// TIA Portal V20 export
// export: Created 2025-12-01T14:57:37.2453598Z, ExportSetting None, DisplayName Totally Integrated Automation Portal, DisplayVersion V20 Update 3, DisplayName TIA Portal Openness, DisplayVersion V20 Update 3, DisplayName TIA Portal Version Control Interface, DisplayVersion V20 Update 3, DisplayName STEP 7 Professional, DisplayVersion V20 Update 3, DisplayName STEP 7 Safety, DisplayVersion V20 Update 2, DisplayName WinCC Basic/Comfort/Advanced, DisplayVersion V20 Update 3, DisplayName WinCC Professional, DisplayVersion V20 Update 3, DisplayName WinCC Unified, DisplayVersion V20 Update 3
FUNCTION_BLOCK "FB74_Presion_DesPaletizadorCajasPlastico"   // FB74, LAD
TITLE = Calculo de la Presion del DesPaletizador de Cajas de Plastico
{ S7_Optimized_Access := 'FALSE' }
// stored: AutoNumber false, SetENOAutomatically false
   VAR_INPUT
      EstadoVI_Mesa : "EstadosMesa";
      EstadoVI_MesaSalida : "EstadosMesa";
      Mesa : UInt;
      MesaSalida : UInt;
      OrdenDesPaletizar : Bool;
      Abierta_PalaMovil : Bool;
      Abriendo_PalaMovil : Bool;
      Cerrando_PalaMovil : Bool;
   END_VAR
   VAR_OUTPUT
      PresionAnalogica : Word;
   END_VAR
   VAR
      TMPInicioPresion : UDInt;
      PresionCalculada : Word;
      MemoPresionSalida : Int;
      CalcularPresion : Bool;
      FinCalcularPresion : Bool;
      RecogerPresion : Bool;
   END_VAR
   VAR_TEMP
      PresionAConvertir : Int;
      PresionSalida : Word;
      PresionDef_Cerrar : Word;
      PresionDef_Abrir : Word;
      PresionInicialCerrar : Int;
      V_TMPInicioPresion : UDInt;
      OK_InicioPresion : Bool;
   END_VAR
   VAR_TEMP   // added for the SCL form of the ladder/FBD networks
      _w1 : Bool;
   END_VAR
BEGIN

REGION Network 1: Incializar
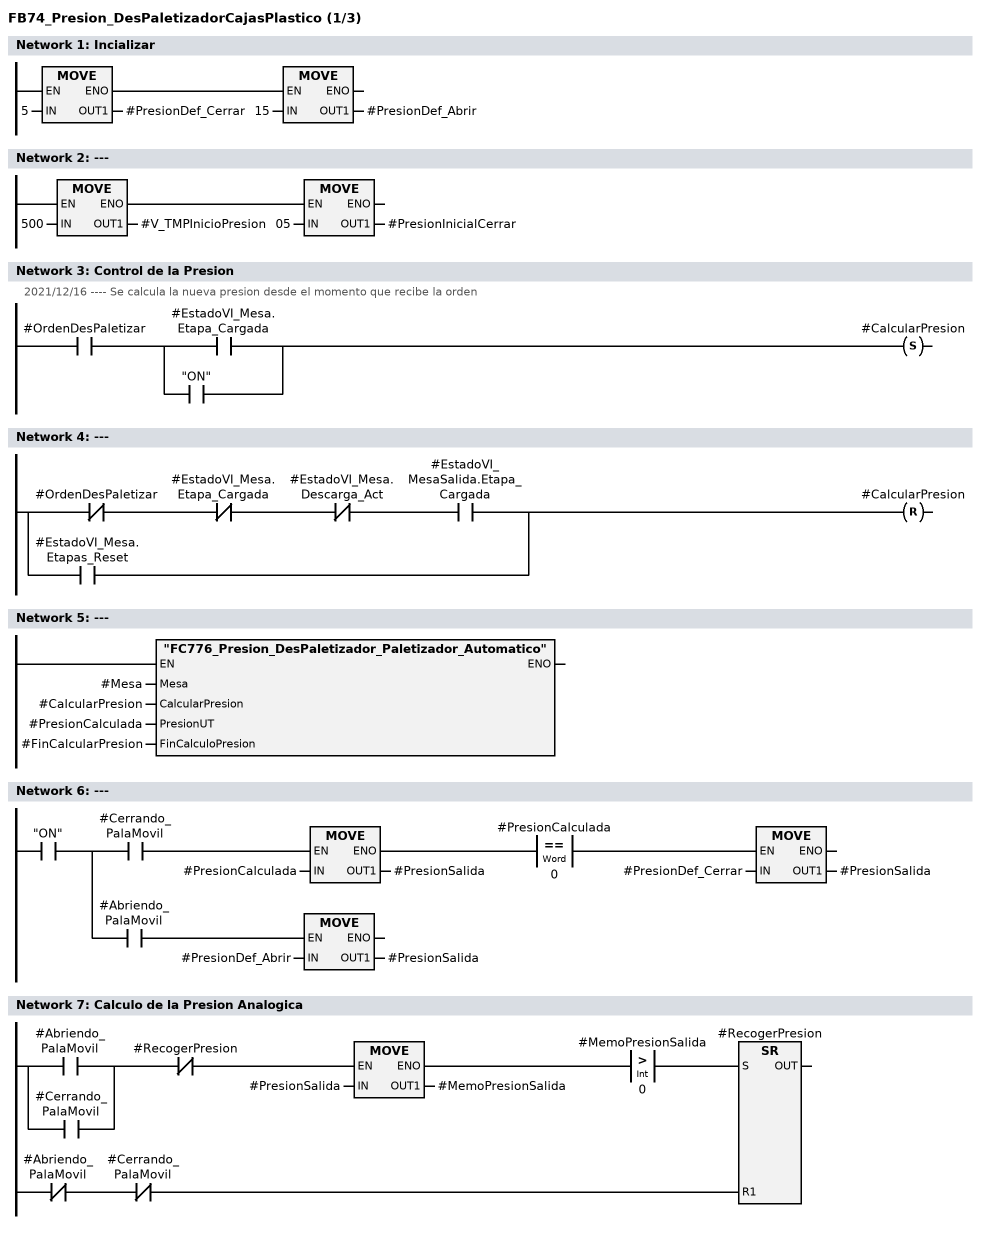
   RUNG wire#powerrail
      { S7_GenerateENO := "TRUE" } Move(in := 5, out1 => #PresionDef_Cerrar)
      { S7_GenerateENO := "TRUE" } Move(in := 15, out1 => #PresionDef_Abrir)
   END_RUNG
   // the same network as SCL:
   // ENO of a box is taken as its EN; it also drops when the box reports an error
   #PresionDef_Cerrar := 5;
   #PresionDef_Abrir := 15;
END_REGION

REGION Network 2: ---
   RUNG wire#powerrail
      { S7_GenerateENO := "TRUE" } Move(in := 500, out1 => #V_TMPInicioPresion)
      { S7_GenerateENO := "TRUE" } Move(in := 05, out1 => #PresionInicialCerrar)
   END_RUNG
   // the same network as SCL:
   // ENO of a box is taken as its EN; it also drops when the box reports an error
   #V_TMPInicioPresion := 500;
   #PresionInicialCerrar := 05;
END_REGION

REGION Network 3: Control de la Presion
   // 2021/12/16 ---- Se calcula la nueva presion desde el momento que recibe la orden
   RUNG wire#powerrail
      Contact( #OrdenDesPaletizar )
      wire#w1
      Contact( #EstadoVI_Mesa.Etapa_Cargada )
      wire#w2
      S_Coil( #CalcularPresion )
   END_RUNG
   RUNG wire#w1
      Contact( "ON" )
   END_RUNG wire#w2
   // the same network as SCL:
   IF #OrdenDesPaletizar AND (#EstadoVI_Mesa.Etapa_Cargada OR "ON") THEN #CalcularPresion := TRUE; END_IF;
END_REGION

REGION Network 4: ---
   RUNG wire#powerrail
      I_Contact( #OrdenDesPaletizar )
      I_Contact( #EstadoVI_Mesa.Etapa_Cargada )
      I_Contact( #EstadoVI_Mesa.Descarga_Act )
      Contact( #EstadoVI_MesaSalida.Etapa_Cargada )
      wire#w1
      R_Coil( #CalcularPresion )
   END_RUNG
   RUNG wire#powerrail
      Contact( #EstadoVI_Mesa.Etapas_Reset )
   END_RUNG wire#w1
   // the same network as SCL:
   IF (NOT #OrdenDesPaletizar AND NOT #EstadoVI_Mesa.Etapa_Cargada AND NOT #EstadoVI_Mesa.Descarga_Act AND #EstadoVI_MesaSalida.Etapa_Cargada) OR #EstadoVI_Mesa.Etapas_Reset THEN
       #CalcularPresion := FALSE;
   END_IF;
END_REGION

REGION Network 5: ---
   RUNG wire#powerrail
      "FC776_Presion_DesPaletizador_Paletizador_Automatico"(Mesa := #Mesa, CalcularPresion := #CalcularPresion, PresionUT := #PresionCalculada, FinCalculoPresion := #FinCalcularPresion)
   END_RUNG
   // the same network as SCL:
   "FC776_Presion_DesPaletizador_Paletizador_Automatico"(Mesa := #Mesa,
                           CalcularPresion := #CalcularPresion,
                           PresionUT := #PresionCalculada,
                           FinCalculoPresion := #FinCalcularPresion);
END_REGION

REGION Network 6: ---
   RUNG wire#powerrail
      Contact( "ON" )
      wire#w1
      Contact( #Cerrando_PalaMovil )
      { S7_GenerateENO := "TRUE" } Move(in := #PresionCalculada, out1 => #PresionSalida)
      { S7_Templates := "SrcType := Word" } EQ_Contact(in1 := #PresionCalculada, in2 := 0)
      { S7_GenerateENO := "TRUE" } Move(in := #PresionDef_Cerrar, out1 => #PresionSalida)
   END_RUNG
   RUNG wire#w1
      Contact( #Abriendo_PalaMovil )
      { S7_GenerateENO := "TRUE" } Move(in := #PresionDef_Abrir, out1 => #PresionSalida)
   END_RUNG
   // the same network as SCL:
   // ENO of a box is taken as its EN; it also drops when the box reports an error
   #_w1 := "ON" AND #Cerrando_PalaMovil;
   IF #_w1 THEN #PresionSalida := #PresionCalculada; END_IF;
   IF #_w1 AND (#PresionCalculada = 0) THEN #PresionSalida := #PresionDef_Cerrar; END_IF;
   IF "ON" AND #Abriendo_PalaMovil THEN #PresionSalida := #PresionDef_Abrir; END_IF;
END_REGION

REGION Network 7: Calculo de la Presion Analogica
   RUNG wire#powerrail
      Contact( #Abriendo_PalaMovil )
      wire#w1
      I_Contact( #RecogerPresion )
      { S7_GenerateENO := "TRUE" } Move(in := #PresionSalida, out1 => #MemoPresionSalida)
      { S7_Templates := "SrcType := Int" } GT_Contact(in1 := #MemoPresionSalida, in2 := 0)
      S_SR(operand := #RecogerPresion, r1 := wire#w2)
   END_RUNG
   RUNG wire#powerrail
      Contact( #Cerrando_PalaMovil )
   END_RUNG wire#w1
   RUNG wire#powerrail
      I_Contact( #Abriendo_PalaMovil )
      I_Contact( #Cerrando_PalaMovil )
   END_RUNG wire#w2
   // the same network as SCL:
   // ENO of a box is taken as its EN; it also drops when the box reports an error
   #_w1 := (#Abriendo_PalaMovil OR #Cerrando_PalaMovil) AND NOT #RecogerPresion;
   IF #_w1 THEN #MemoPresionSalida := #PresionSalida; END_IF;
   IF #_w1 AND (#MemoPresionSalida > 0) THEN
       #RecogerPresion := TRUE;   // SR flip-flop
   END_IF;
   IF NOT #Abriendo_PalaMovil AND NOT #Cerrando_PalaMovil THEN #RecogerPresion := FALSE; END_IF;
END_REGION

REGION Network 8: Presion de Salida
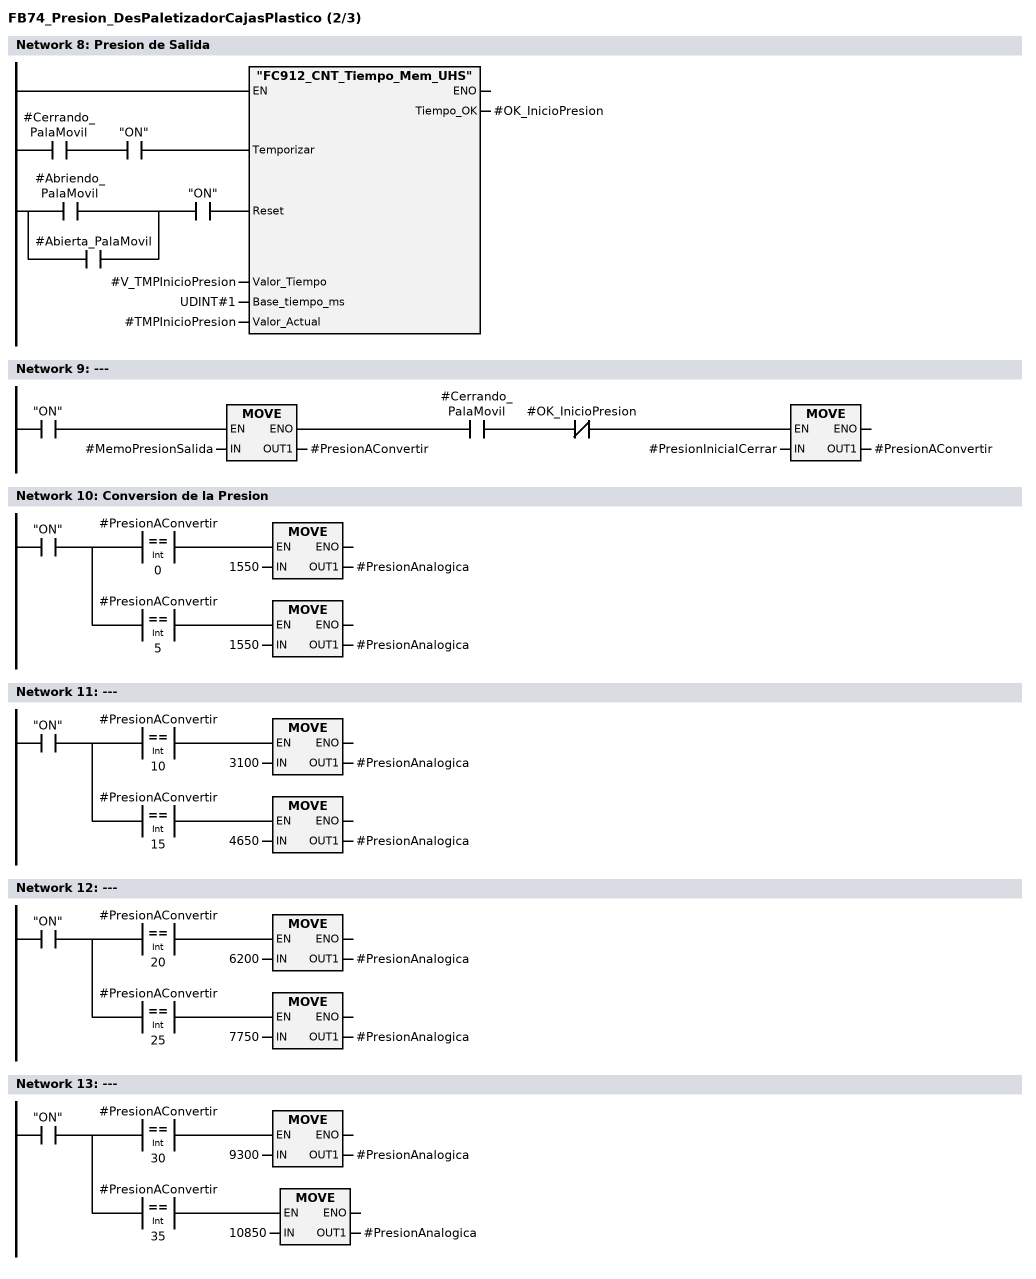
   RUNG wire#powerrail
      "FC912_CNT_Tiempo_Mem_UHS"(Temporizar := wire#w1, Reset := wire#w3, Valor_Tiempo := #V_TMPInicioPresion, Base_tiempo_ms := UDINT#1, Valor_Actual := #TMPInicioPresion, Tiempo_OK => #OK_InicioPresion)
   END_RUNG
   RUNG wire#powerrail
      Contact( #Cerrando_PalaMovil )
      Contact( "ON" )
   END_RUNG wire#w1
   RUNG wire#powerrail
      Contact( #Abriendo_PalaMovil )
      wire#w2
      Contact( "ON" )
   END_RUNG wire#w3
   RUNG wire#powerrail
      Contact( #Abierta_PalaMovil )
   END_RUNG wire#w2
   // the same network as SCL:
   "FC912_CNT_Tiempo_Mem_UHS"(Temporizar := #Cerrando_PalaMovil AND "ON",
                           Reset := (#Abriendo_PalaMovil OR #Abierta_PalaMovil) AND "ON",
                           Valor_Tiempo := #V_TMPInicioPresion,
                           Base_tiempo_ms := UDINT#1,
                           Valor_Actual := #TMPInicioPresion,
                           Tiempo_OK => #OK_InicioPresion);
END_REGION

REGION Network 9: ---
   RUNG wire#powerrail
      Contact( "ON" )
      { S7_GenerateENO := "TRUE" } Move(in := #MemoPresionSalida, out1 => #PresionAConvertir)
      Contact( #Cerrando_PalaMovil )
      I_Contact( #OK_InicioPresion )
      { S7_GenerateENO := "TRUE" } Move(in := #PresionInicialCerrar, out1 => #PresionAConvertir)
   END_RUNG
   // the same network as SCL:
   // ENO of a box is taken as its EN; it also drops when the box reports an error
   IF "ON" THEN #PresionAConvertir := #MemoPresionSalida; END_IF;
   IF "ON" AND #Cerrando_PalaMovil AND NOT #OK_InicioPresion THEN
       #PresionAConvertir := #PresionInicialCerrar;
   END_IF;
END_REGION

REGION Network 10: Conversion de la Presion
   RUNG wire#powerrail
      Contact( "ON" )
      wire#w1
      { S7_Templates := "SrcType := Int" } EQ_Contact(in1 := #PresionAConvertir, in2 := 0)
      { S7_GenerateENO := "TRUE" } Move(in := 1550, out1 => #PresionAnalogica)
   END_RUNG
   RUNG wire#w1
      { S7_Templates := "SrcType := Int" } EQ_Contact(in1 := #PresionAConvertir, in2 := 5)
      { S7_GenerateENO := "TRUE" } Move(in := 1550, out1 => #PresionAnalogica)
   END_RUNG
   // the same network as SCL:
   IF "ON" AND (#PresionAConvertir = 0) THEN #PresionAnalogica := 1550; END_IF;
   IF "ON" AND (#PresionAConvertir = 5) THEN #PresionAnalogica := 1550; END_IF;
END_REGION

REGION Network 11: ---
   RUNG wire#powerrail
      Contact( "ON" )
      wire#w1
      { S7_Templates := "SrcType := Int" } EQ_Contact(in1 := #PresionAConvertir, in2 := 10)
      { S7_GenerateENO := "TRUE" } Move(in := 3100, out1 => #PresionAnalogica)
   END_RUNG
   RUNG wire#w1
      { S7_Templates := "SrcType := Int" } EQ_Contact(in1 := #PresionAConvertir, in2 := 15)
      { S7_GenerateENO := "TRUE" } Move(in := 4650, out1 => #PresionAnalogica)
   END_RUNG
   // the same network as SCL:
   IF "ON" AND (#PresionAConvertir = 10) THEN #PresionAnalogica := 3100; END_IF;
   IF "ON" AND (#PresionAConvertir = 15) THEN #PresionAnalogica := 4650; END_IF;
END_REGION

REGION Network 12: ---
   RUNG wire#powerrail
      Contact( "ON" )
      wire#w1
      { S7_Templates := "SrcType := Int" } EQ_Contact(in1 := #PresionAConvertir, in2 := 20)
      { S7_GenerateENO := "TRUE" } Move(in := 6200, out1 => #PresionAnalogica)
   END_RUNG
   RUNG wire#w1
      { S7_Templates := "SrcType := Int" } EQ_Contact(in1 := #PresionAConvertir, in2 := 25)
      { S7_GenerateENO := "TRUE" } Move(in := 7750, out1 => #PresionAnalogica)
   END_RUNG
   // the same network as SCL:
   IF "ON" AND (#PresionAConvertir = 20) THEN #PresionAnalogica := 6200; END_IF;
   IF "ON" AND (#PresionAConvertir = 25) THEN #PresionAnalogica := 7750; END_IF;
END_REGION

REGION Network 13: ---
   RUNG wire#powerrail
      Contact( "ON" )
      wire#w1
      { S7_Templates := "SrcType := Int" } EQ_Contact(in1 := #PresionAConvertir, in2 := 30)
      { S7_GenerateENO := "TRUE" } Move(in := 9300, out1 => #PresionAnalogica)
   END_RUNG
   RUNG wire#w1
      { S7_Templates := "SrcType := Int" } EQ_Contact(in1 := #PresionAConvertir, in2 := 35)
      { S7_GenerateENO := "TRUE" } Move(in := 10850, out1 => #PresionAnalogica)
   END_RUNG
   // the same network as SCL:
   IF "ON" AND (#PresionAConvertir = 30) THEN #PresionAnalogica := 9300; END_IF;
   IF "ON" AND (#PresionAConvertir = 35) THEN #PresionAnalogica := 10850; END_IF;
END_REGION

REGION Network 14: ---
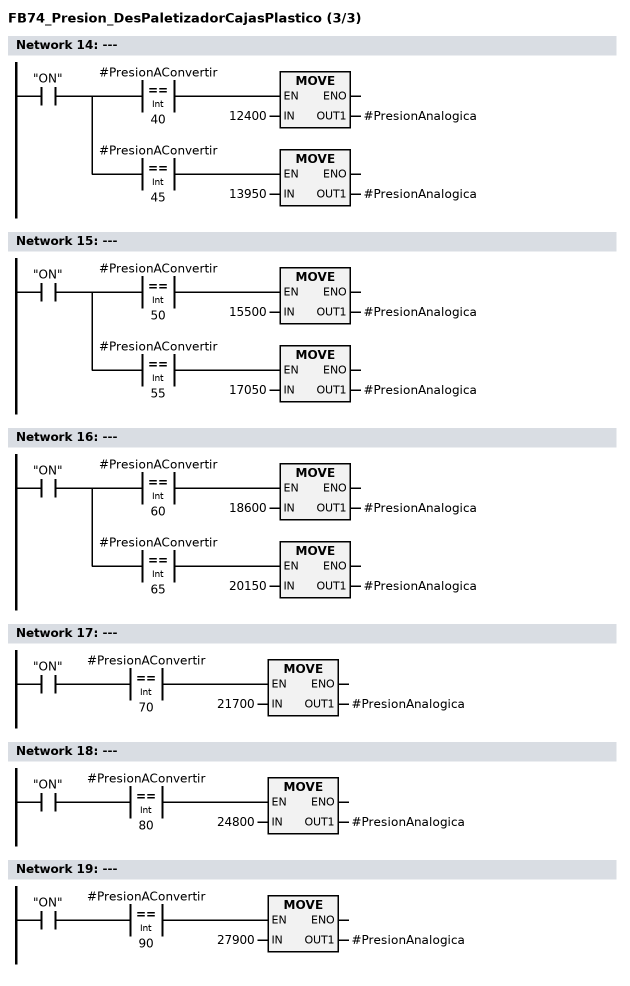
   RUNG wire#powerrail
      Contact( "ON" )
      wire#w1
      { S7_Templates := "SrcType := Int" } EQ_Contact(in1 := #PresionAConvertir, in2 := 40)
      { S7_GenerateENO := "TRUE" } Move(in := 12400, out1 => #PresionAnalogica)
   END_RUNG
   RUNG wire#w1
      { S7_Templates := "SrcType := Int" } EQ_Contact(in1 := #PresionAConvertir, in2 := 45)
      { S7_GenerateENO := "TRUE" } Move(in := 13950, out1 => #PresionAnalogica)
   END_RUNG
   // the same network as SCL:
   IF "ON" AND (#PresionAConvertir = 40) THEN #PresionAnalogica := 12400; END_IF;
   IF "ON" AND (#PresionAConvertir = 45) THEN #PresionAnalogica := 13950; END_IF;
END_REGION

REGION Network 15: ---
   RUNG wire#powerrail
      Contact( "ON" )
      wire#w1
      { S7_Templates := "SrcType := Int" } EQ_Contact(in1 := #PresionAConvertir, in2 := 50)
      { S7_GenerateENO := "TRUE" } Move(in := 15500, out1 => #PresionAnalogica)
   END_RUNG
   RUNG wire#w1
      { S7_Templates := "SrcType := Int" } EQ_Contact(in1 := #PresionAConvertir, in2 := 55)
      { S7_GenerateENO := "TRUE" } Move(in := 17050, out1 => #PresionAnalogica)
   END_RUNG
   // the same network as SCL:
   IF "ON" AND (#PresionAConvertir = 50) THEN #PresionAnalogica := 15500; END_IF;
   IF "ON" AND (#PresionAConvertir = 55) THEN #PresionAnalogica := 17050; END_IF;
END_REGION

REGION Network 16: ---
   RUNG wire#powerrail
      Contact( "ON" )
      wire#w1
      { S7_Templates := "SrcType := Int" } EQ_Contact(in1 := #PresionAConvertir, in2 := 60)
      { S7_GenerateENO := "TRUE" } Move(in := 18600, out1 => #PresionAnalogica)
   END_RUNG
   RUNG wire#w1
      { S7_Templates := "SrcType := Int" } EQ_Contact(in1 := #PresionAConvertir, in2 := 65)
      { S7_GenerateENO := "TRUE" } Move(in := 20150, out1 => #PresionAnalogica)
   END_RUNG
   // the same network as SCL:
   IF "ON" AND (#PresionAConvertir = 60) THEN #PresionAnalogica := 18600; END_IF;
   IF "ON" AND (#PresionAConvertir = 65) THEN #PresionAnalogica := 20150; END_IF;
END_REGION

REGION Network 17: ---
   RUNG wire#powerrail
      Contact( "ON" )
      { S7_Templates := "SrcType := Int" } EQ_Contact(in1 := #PresionAConvertir, in2 := 70)
      { S7_GenerateENO := "TRUE" } Move(in := 21700, out1 => #PresionAnalogica)
   END_RUNG
   // the same network as SCL:
   IF "ON" AND (#PresionAConvertir = 70) THEN #PresionAnalogica := 21700; END_IF;
END_REGION

REGION Network 18: ---
   RUNG wire#powerrail
      Contact( "ON" )
      { S7_Templates := "SrcType := Int" } EQ_Contact(in1 := #PresionAConvertir, in2 := 80)
      { S7_GenerateENO := "TRUE" } Move(in := 24800, out1 => #PresionAnalogica)
   END_RUNG
   // the same network as SCL:
   IF "ON" AND (#PresionAConvertir = 80) THEN #PresionAnalogica := 24800; END_IF;
END_REGION

REGION Network 19: ---
   RUNG wire#powerrail
      Contact( "ON" )
      { S7_Templates := "SrcType := Int" } EQ_Contact(in1 := #PresionAConvertir, in2 := 90)
      { S7_GenerateENO := "TRUE" } Move(in := 27900, out1 => #PresionAnalogica)
   END_RUNG
   // the same network as SCL:
   IF "ON" AND (#PresionAConvertir = 90) THEN #PresionAnalogica := 27900; END_IF;
END_REGION
END_FUNCTION_BLOCK
